KUKA KRL data list: TPadraoSTR.dat

&ACCESS RV2
DEFDAT TPadraoSTR
   INT  I,J,k
ENDDAT
